Staubli VAL3: start.pgx

program start()
begin

  userPage("pala_cinke")
  call cakajProgress(1)
  enablePower()
  setMonitorSpeed(50)

  taskCreate "Safety",80,safety()

  movej(pHome,flange,mSrednje)

  // Ali robot izvaja (pekalni) task
  nTaskWorking = 0
  // Čas peke (Čas1 = čas pečenja na prvi strani)
  nCas_peke1=95
  nCas_peke2=nCas_peke1*0.8

  do
    jTrenutna=herej()
  until false
end
